TEXTLIST TL_E_INSTANCE_CMD
  0 = 'NULL'
  1 = 'INIT'
  2 = 'DISABLE'
  3 = 'ENABLE'
  4 = 'WORK'
  102 = 'CLEAR'
   = ''
END_TEXTLIST

(* stored: Version 1.1.0.1, ProductVersion 3.1.4024.15
   TextList TL_E_INSTANCE_CMD: Id {558d2c0e-5c3a-4624-bb10-83ff7ef138ab} *)
